{attribute 'GeneratedUsingTerminal: EL6022-0000-0016'}
{attribute addProperty BoxType "EL6022-0000-0016"}
{attribute addProperty Description "EL6022 Interface 2Ch. (RS422/485)"}
{attribute addProperty Physics "KK"}
{attribute addProperty Id "COM_Inputs_Channel_1AT %I*COM_Inputs_Channel_3801C95E30COM_Inputs_Channel_2AT %I*COM_Inputs_Channel_3801C95E30COM_Outputs_Channel_1AT %Q*COM_Outputs_Channel_EADA2E0D27COM_Outputs_Channel_2AT %Q*COM_Outputs_Channel_EADA2E0D27WcStateAT %I*WcState_9091E0EB2InfoDataAT %I*InfoData_32EB74EA10"}
{attribute addProperty CRC "3585370301"}
{attribute addProperty Size "126"}
TYPE EL6022_D5B468BD EXTENDS EtcSlaveTerminalBase_947E5A46 :
STRUCT
	{attribute addProperty Name "COM_Inputs_Channel_1"}
	COM_Inputs_Channel_1 : COM_Inputs_Channel_3801C95E;
	{attribute addProperty Name "COM_Inputs_Channel_2"}
	COM_Inputs_Channel_2 : COM_Inputs_Channel_3801C95E;
	{attribute addProperty Name "COM_Outputs_Channel_1"}
	COM_Outputs_Channel_1 : COM_Outputs_Channel_EADA2E0D;
	{attribute addProperty Name "COM_Outputs_Channel_2"}
	COM_Outputs_Channel_2 : COM_Outputs_Channel_EADA2E0D;
	{attribute addProperty Name "WcState"}
	WcState : WcState_9091E0EB;
	{attribute addProperty Name "InfoData"}
	InfoData : InfoData_32EB74EA;
END_STRUCT
END_TYPE

(* stored: Version 1.2.0.0, ProductVersion 3.1.4024.9
   DUT EL6022_D5B468BD: Id {6211b075-955a-460c-bd9a-30d8759d5c9c} *)
